INTERFACE I_DisSensor

PROPERTY Distance : LREAL
GET
END_GET
END_PROPERTY

END_INTERFACE

(* stored: Version 1.1.0.1, ProductVersion 3.1.4026.13
   Itf I_DisSensor: Id {3e654df5-60d0-499f-a6da-635647f372fc}
   Property Distance: Id {74771d1d-c132-4373-9d42-75faa42f8ee0}
   Get Get: Id {5dd6e67d-66a4-4637-a081-88b4b864db7b} *)
